FUNCTION_BLOCK E_PERMIT_1 (* Permissive propagation of 1 event channel (generic FB) *)
  (* Standard: 61499-1 Annex A; Description: Copyright (c) 2026 Meisterschulen am Ostbahnhof This program and the accompanying materials are made available under the terms of the Eclipse Public License 2.0 which is available at https://www.eclipse.org/legal/epl-2.0/ SPDX-License-Identifier: EPL-2.0 *)
  (* Version 3.0, 2025-04-14, Patrick Aigner, changed package *)
  (* Version 1.0, 2026-09-10, Franz Höpfinger, Meisterschulen am Ostbahnhof, initial implementation *)
  PACKAGE iec61499::events;
  {SET_ATTRIBUTE(eclipse4diac::core::GenericClassName, 'GEN_E_PERMIT')}
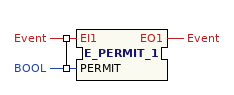
  EVENT_INPUT
    EI1 WITH PERMIT; (* Event input channel 1 *)
  END_EVENT
  EVENT_OUTPUT
    EO1; (* Event output channel 1 *)
  END_EVENT
  VAR_INPUT
    PERMIT : BOOL; (* Permit condition *)
  END_VAR
END_FUNCTION_BLOCK
